// TIA Portal V15.1 export
// export: Created 2024-06-21T08:40:55.8760909Z, ExportSetting WithDefaults, DisplayName Totally Integrated Automation Portal, DisplayVersion V15.1 Update 5, DisplayName TIA Portal Openness, DisplayVersion V15.1 Update 5, DisplayName SINAMICS Startdrive Advanced, DisplayVersion V15.1, DisplayName G130, G150, S120, S150, SINAMICS MV, S210, DisplayVersion V15.1, DisplayName G110M, G120, G120C, G120D, G120P, DisplayVersion V15.1, DisplayName STEP 7 Professional, DisplayVersion V15.1 Update 5, DisplayName STEP 7 Safety, DisplayVersion V15.1, DisplayName WinCC Professional, DisplayVersion V15.1 Update 5, DisplayName SIMATIC Visualization Architect, DisplayVersion V15.1
FUNCTION "LVD-Config" : Void   // FC1910, FBD
TITLE = LVDConfig
{ S7_Optimized_Access := 'TRUE' }
AUTHOR : VCC
FAMILY : Config
VERSION : 0.1
// =============================================================================
// VD Communication Configuration
// =============================================================================
// stored: AutoNumber false, IsIECCheckEnabled false, SetENOAutomatically False, UDAEnableTagReadback false
   VAR_INPUT
      C_ConnId : Int;   // Connection identification
      C_IpAdress1 : Int;   // IP adress byte 1
      C_IpAdress2 : Int;   // IP adress byte 2
      C_IpAdress3 : Int;   // IP adress byte 3
      C_IpAdress4 : Int;   // IP adress byte 4
      C_DeviceID : Int;   // 1 = ET200S, 2=315/317, 3 = 319 / Device ID
      C_Active : Bool;   // Yes = this machine connects actively
   END_VAR
   VAR_IN_OUT
      IO_VDConfig : TCON_Param;   // VD configuration DB / VD configuration
   END_VAR
   VAR_TEMP
      RemoteAddressLen : Int;   // Number Of Bytes Defining The Remote IP Address
   END_VAR
BEGIN

REGION Network 1: **** 1 - Inputs **** Init Values
   // Init Values
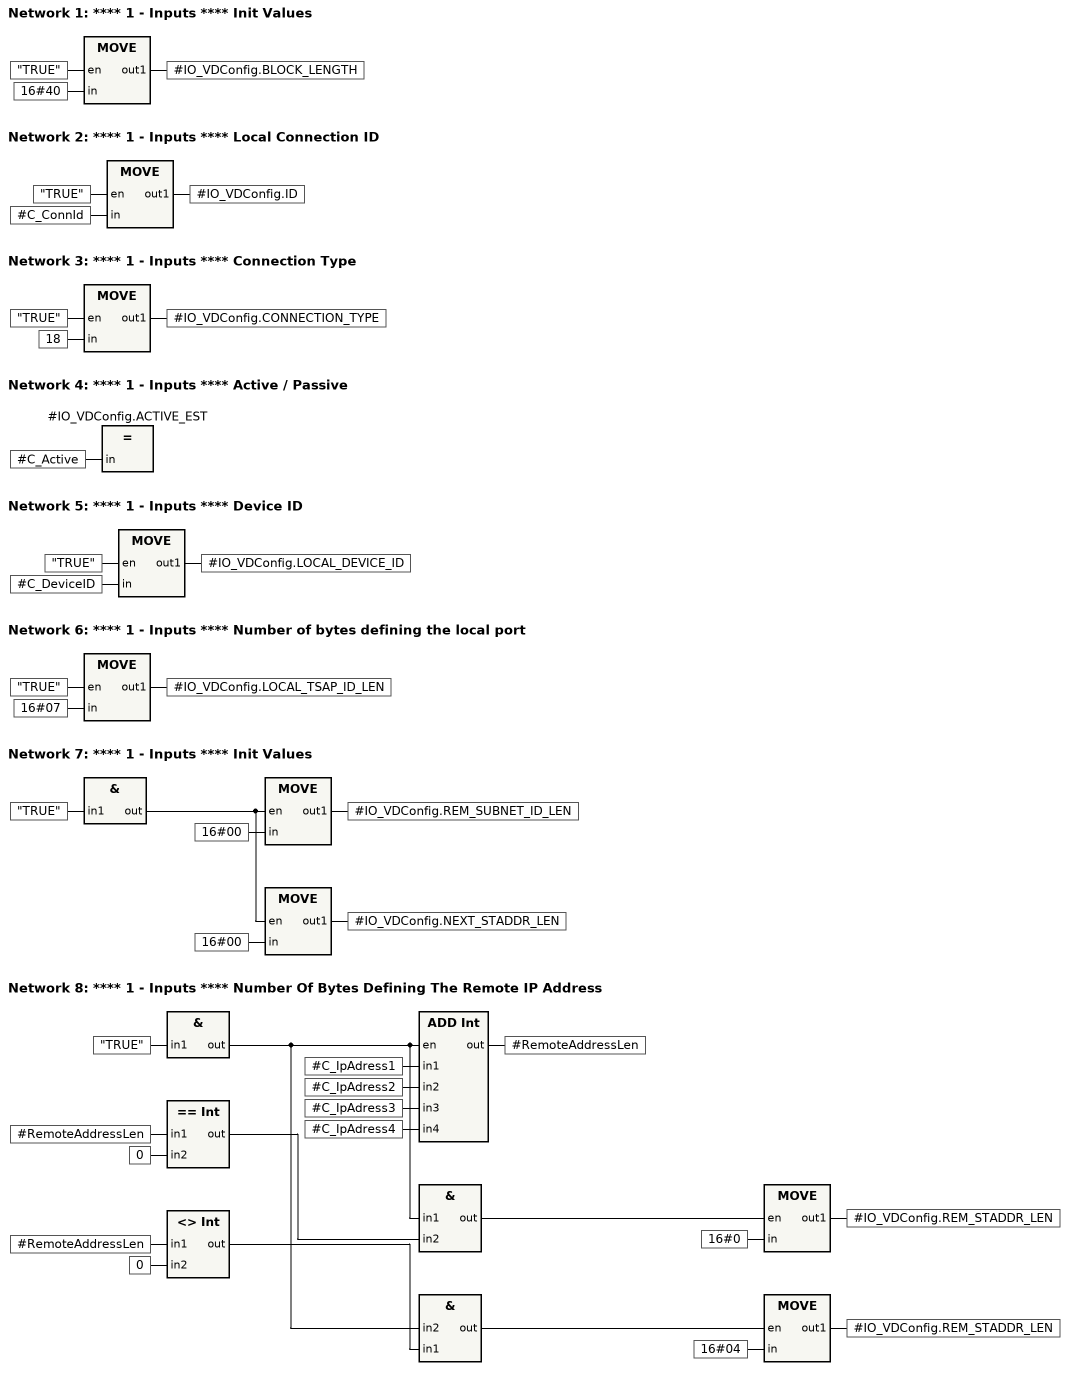
   IF "TRUE" THEN #IO_VDConfig.BLOCK_LENGTH := 16#40; END_IF;
END_REGION

REGION Network 2: **** 1 - Inputs **** Local Connection ID
   // Local Connection ID
   IF "TRUE" THEN #IO_VDConfig.ID := #C_ConnId; END_IF;
END_REGION

REGION Network 3: **** 1 - Inputs **** Connection Type
   // Connection Type
   IF "TRUE" THEN #IO_VDConfig.CONNECTION_TYPE := 18; END_IF;
END_REGION

REGION Network 4: **** 1 - Inputs **** Active / Passive
   // Active / Passive
   #IO_VDConfig.ACTIVE_EST := #C_Active;
END_REGION

REGION Network 5: **** 1 - Inputs **** Device ID
   // Device ID
   IF "TRUE" THEN #IO_VDConfig.LOCAL_DEVICE_ID := #C_DeviceID; END_IF;
END_REGION

REGION Network 6: **** 1 - Inputs **** Number of bytes defining the local port
   // Number of bytes defining the local port
   IF "TRUE" THEN #IO_VDConfig.LOCAL_TSAP_ID_LEN := 16#07; END_IF;
END_REGION

REGION Network 7: **** 1 - Inputs **** Init Values
   // Init Values
   IF "TRUE" THEN
       #IO_VDConfig.REM_SUBNET_ID_LEN := 16#00;
       #IO_VDConfig.NEXT_STADDR_LEN := 16#00;
   END_IF;
END_REGION

REGION Network 8: **** 1 - Inputs **** Number Of Bytes Defining The Remote IP Address
   // Number Of Bytes Defining The Remote IP Address
   IF "TRUE" THEN #RemoteAddressLen := #C_IpAdress1 + #C_IpAdress2 + #C_IpAdress3 + #C_IpAdress4; END_IF;
   IF "TRUE" AND (#RemoteAddressLen = 0) THEN #IO_VDConfig.REM_STADDR_LEN := 16#0; END_IF;
   IF "TRUE" AND (#RemoteAddressLen <> 0) THEN #IO_VDConfig.REM_STADDR_LEN := 16#04; END_IF;
END_REGION

REGION Network 9: **** 1 - Inputs **** Remote ID Length
   // Remote ID Length
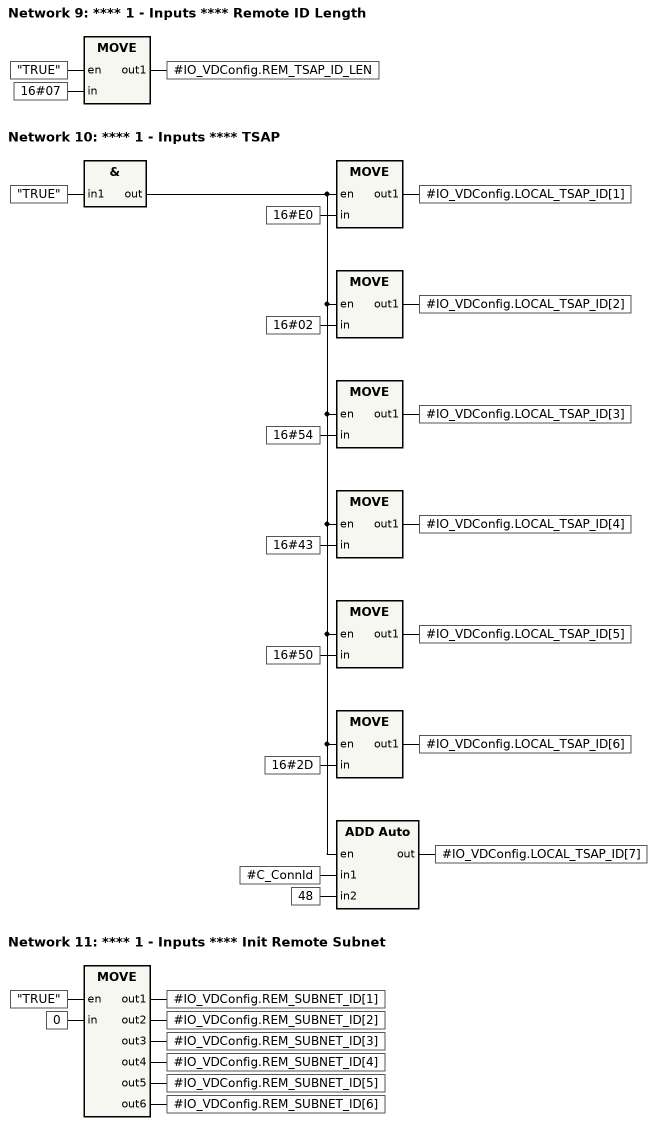
   IF "TRUE" THEN #IO_VDConfig.REM_TSAP_ID_LEN := 16#07; END_IF;
END_REGION

REGION Network 10: **** 1 - Inputs **** TSAP
   // TSAP
   IF "TRUE" THEN
       #IO_VDConfig.LOCAL_TSAP_ID[1] := 16#E0;
       #IO_VDConfig.LOCAL_TSAP_ID[2] := 16#02;
       #IO_VDConfig.LOCAL_TSAP_ID[3] := 16#54;
       #IO_VDConfig.LOCAL_TSAP_ID[4] := 16#43;
       #IO_VDConfig.LOCAL_TSAP_ID[5] := 16#50;
       #IO_VDConfig.LOCAL_TSAP_ID[6] := 16#2D;
       #IO_VDConfig.LOCAL_TSAP_ID[7] := #C_ConnId + 48;
   END_IF;
END_REGION

REGION Network 11: **** 1 - Inputs **** Init Remote Subnet
   // Init Remote Subnet
   IF "TRUE" THEN
       #IO_VDConfig.REM_SUBNET_ID[1] := 0;
       #IO_VDConfig.REM_SUBNET_ID[2] := 0;
       #IO_VDConfig.REM_SUBNET_ID[3] := 0;
       #IO_VDConfig.REM_SUBNET_ID[4] := 0;
       #IO_VDConfig.REM_SUBNET_ID[5] := 0;
       #IO_VDConfig.REM_SUBNET_ID[6] := 0;
   END_IF;
END_REGION

REGION Network 12: **** 1 - Inputs **** Remote IP Address
   // Remote IP Address
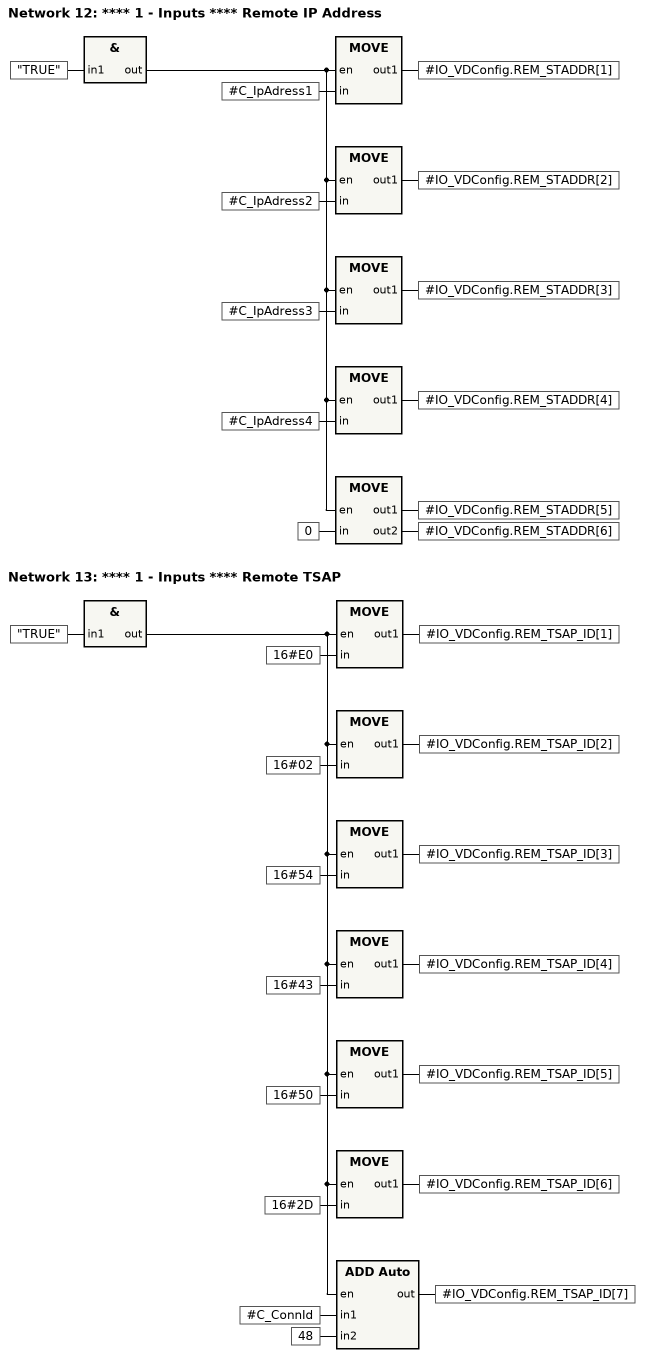
   IF "TRUE" THEN
       #IO_VDConfig.REM_STADDR[1] := #C_IpAdress1;
       #IO_VDConfig.REM_STADDR[2] := #C_IpAdress2;
       #IO_VDConfig.REM_STADDR[3] := #C_IpAdress3;
       #IO_VDConfig.REM_STADDR[4] := #C_IpAdress4;
       #IO_VDConfig.REM_STADDR[5] := 0;
       #IO_VDConfig.REM_STADDR[6] := 0;
   END_IF;
END_REGION

REGION Network 13: **** 1 - Inputs **** Remote TSAP
   // Remote TSAP
   IF "TRUE" THEN
       #IO_VDConfig.REM_TSAP_ID[1] := 16#E0;
       #IO_VDConfig.REM_TSAP_ID[2] := 16#02;
       #IO_VDConfig.REM_TSAP_ID[3] := 16#54;
       #IO_VDConfig.REM_TSAP_ID[4] := 16#43;
       #IO_VDConfig.REM_TSAP_ID[5] := 16#50;
       #IO_VDConfig.REM_TSAP_ID[6] := 16#2D;
       #IO_VDConfig.REM_TSAP_ID[7] := #C_ConnId + 48;
   END_IF;
END_REGION
END_FUNCTION
